// TIA Portal V18 export
FUNCTION "_motionLevel0_axis_main_in_cyclic_interrupt" : Void   // FC13, FBD
{ S7_Optimized_Access := 'TRUE' }
VERSION : 0.1
// stored: AutoNumber true, IsIECCheckEnabled false, SetENOAutomatically false, UDAEnableTagReadback false
   VAR_TEMP
      doors : Bool;
      "xray uses doors fwd closed mech" : Bool;
      "добавить блокировку вперед по световой завесе" : Bool;
      loc_dor_c_opn : Bool;
      loc_dor_c_cls : Bool;
      doorsWnOpnNAld : Bool;
      doorsWnClsNAld : Bool;
      ошибка_задания_искуственных_границ : Bool;
      динамическая_граница_y_rev : Real;
      динамическая_граница_y_fwd : Real;
      динамическая_граница_x_rev : Real;
      динамическая_граница_x_fwd : Real;
      манипулятор_не_мешает_дверям : Bool;
      doors_wnmanipulator : Bool;
   END_VAR
BEGIN

REGION Network 2
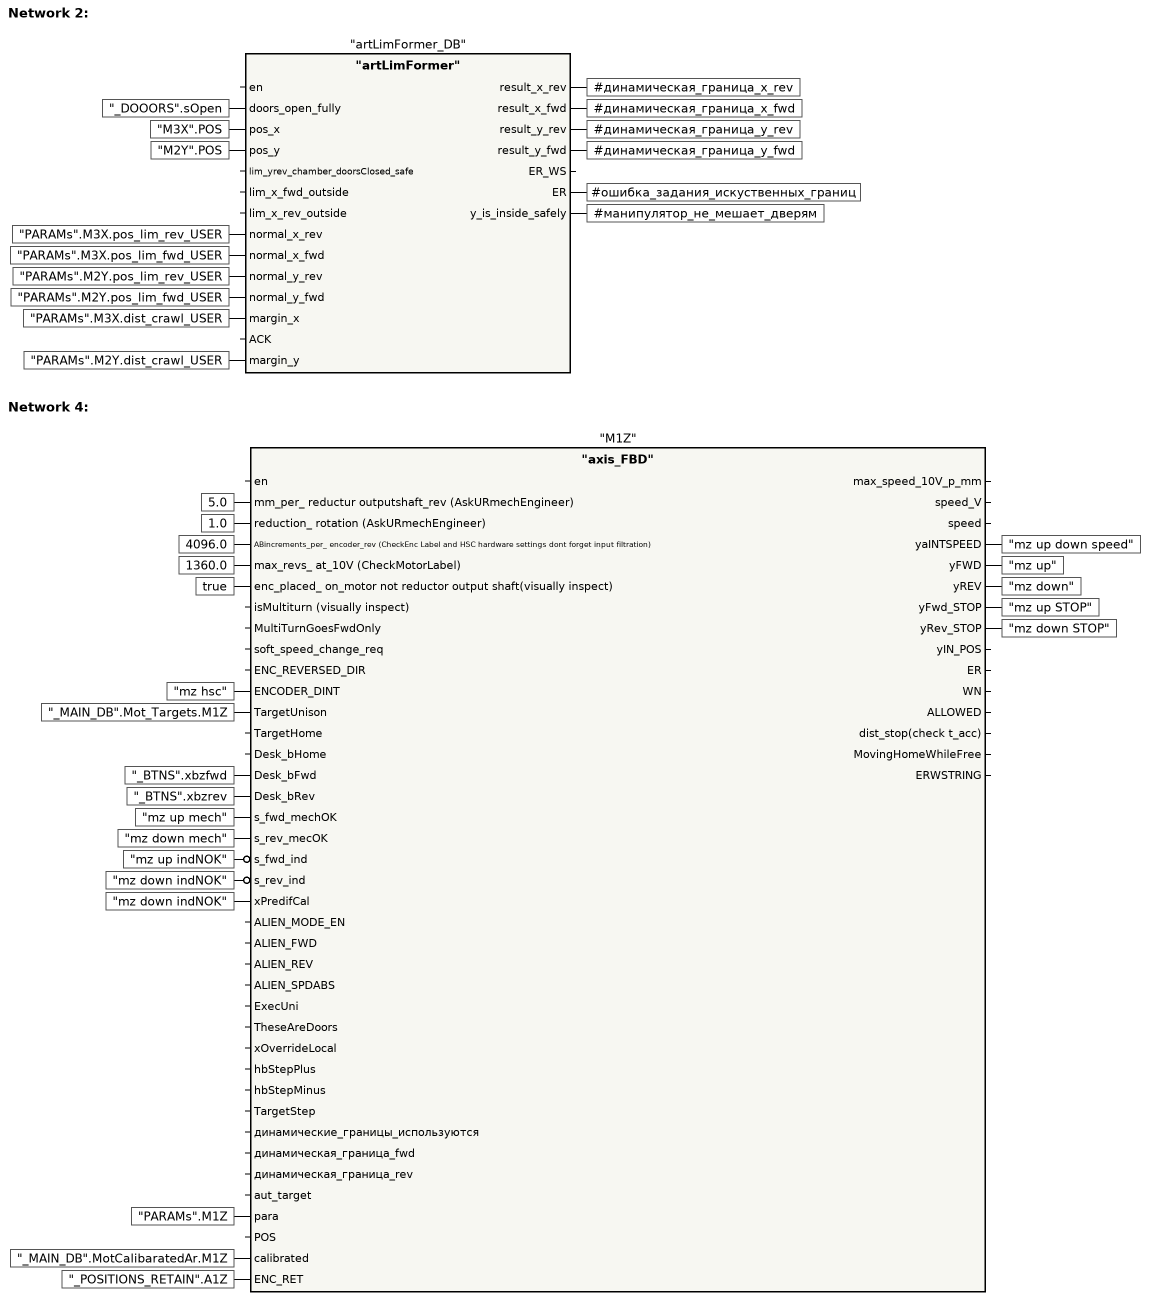
   "artLimFormer_DB"(doors_open_fully := "_DOOORS".sOpen,   // "artLimFormer"
                     pos_x := "M3X".POS,
                     pos_y := "M2Y".POS,
                     normal_x_rev := "PARAMs".M3X.pos_lim_rev_USER,
                     normal_x_fwd := "PARAMs".M3X.pos_lim_fwd_USER,
                     normal_y_rev := "PARAMs".M2Y.pos_lim_rev_USER,
                     normal_y_fwd := "PARAMs".M2Y.pos_lim_fwd_USER,
                     margin_x := "PARAMs".M3X.dist_crawl_USER,
                     margin_y := "PARAMs".M2Y.dist_crawl_USER,
                     result_x_rev => #динамическая_граница_x_rev,
                     result_x_fwd => #динамическая_граница_x_fwd,
                     result_y_rev => #динамическая_граница_y_rev,
                     result_y_fwd => #динамическая_граница_y_fwd,
                     ER => #ошибка_задания_искуственных_границ,
                     y_is_inside_safely => #манипулятор_не_мешает_дверям);
END_REGION

REGION Network 4
   "M1Z"("mm_per_ reductur outputshaft_rev (AskURmechEngineer)" := 5.0,   // "axis_FBD"
         "reduction_ rotation (AskURmechEngineer)" := 1.0,
         "ABincrements_per_ encoder_rev (CheckEnc Label and HSC hardware settings dont forget input filtration)" := 4096.0,
         "max_revs_ at_10V (CheckMotorLabel)" := 1360.0,
         "enc_placed_ on_motor not reductor output shaft(visually inspect)" := true,
         ENCODER_DINT := "mz hsc",
         TargetUnison := "_MAIN_DB".Mot_Targets.M1Z,
         Desk_bFwd := "_BTNS".xbzfwd,
         Desk_bRev := "_BTNS".xbzrev,
         s_fwd_mechOK := "mz up mech",
         s_rev_mecOK := "mz down mech",
         s_fwd_ind := NOT "mz up indNOK",
         s_rev_ind := NOT "mz down indNOK",
         xPredifCal := "mz down indNOK",
         para := "PARAMs".M1Z,
         calibrated := "_MAIN_DB".MotCalibaratedAr.M1Z,
         ENC_RET := "_POSITIONS_RETAIN".A1Z,
         yaINTSPEED => "mz up down speed",
         yFWD => "mz up",
         yREV => "mz down",
         yFwd_STOP => "mz up STOP",
         yRev_STOP => "mz down STOP");
END_REGION

REGION Network 5
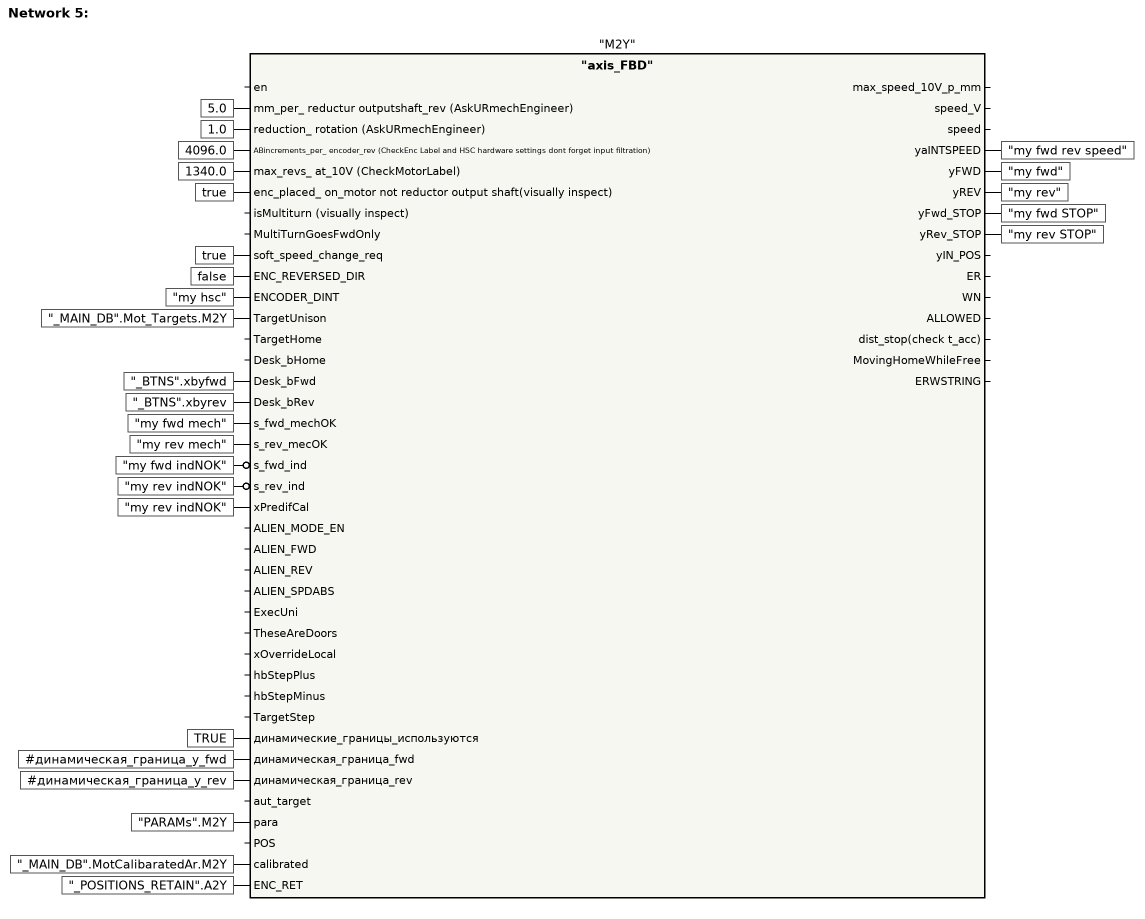
   "M2Y"("mm_per_ reductur outputshaft_rev (AskURmechEngineer)" := 5.0,   // "axis_FBD"
         "reduction_ rotation (AskURmechEngineer)" := 1.0,
         "ABincrements_per_ encoder_rev (CheckEnc Label and HSC hardware settings dont forget input filtration)" := 4096.0,
         "max_revs_ at_10V (CheckMotorLabel)" := 1340.0,
         "enc_placed_ on_motor not reductor output shaft(visually inspect)" := true,
         soft_speed_change_req := true,
         ENC_REVERSED_DIR := false,
         ENCODER_DINT := "my hsc",
         TargetUnison := "_MAIN_DB".Mot_Targets.M2Y,
         Desk_bFwd := "_BTNS".xbyfwd,
         Desk_bRev := "_BTNS".xbyrev,
         s_fwd_mechOK := "my fwd mech",
         s_rev_mecOK := "my rev mech",
         s_fwd_ind := NOT "my fwd indNOK",
         s_rev_ind := NOT "my rev indNOK",
         xPredifCal := "my rev indNOK",
         динамические_границы_используются := TRUE,
         динамическая_граница_fwd := #динамическая_граница_y_fwd,
         динамическая_граница_rev := #динамическая_граница_y_rev,
         para := "PARAMs".M2Y,
         calibrated := "_MAIN_DB".MotCalibaratedAr.M2Y,
         ENC_RET := "_POSITIONS_RETAIN".A2Y,
         yaINTSPEED => "my fwd rev speed",
         yFWD => "my fwd",
         yREV => "my rev",
         yFwd_STOP => "my fwd STOP",
         yRev_STOP => "my rev STOP");
END_REGION

REGION Network 6
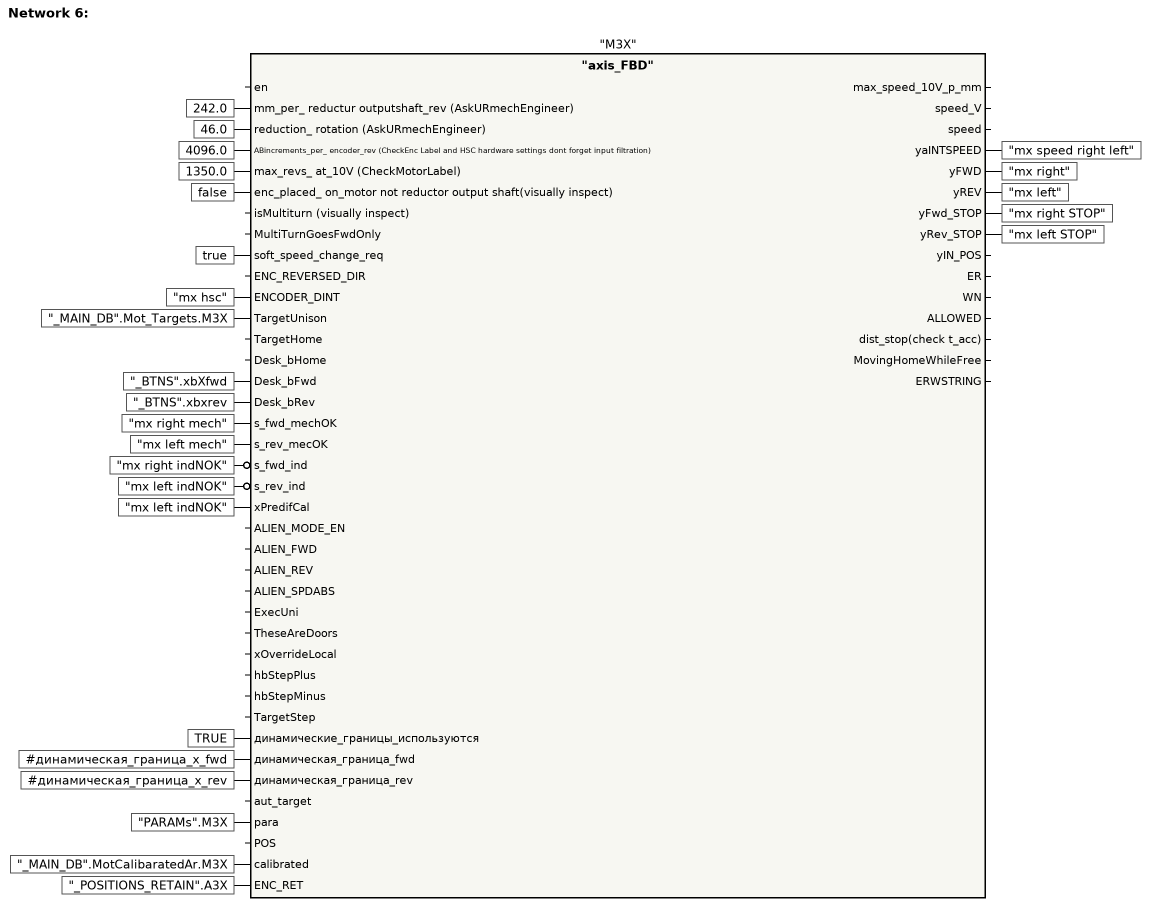
   "M3X"("mm_per_ reductur outputshaft_rev (AskURmechEngineer)" := 242.0,   // "axis_FBD"
         "reduction_ rotation (AskURmechEngineer)" := 46.0,
         "ABincrements_per_ encoder_rev (CheckEnc Label and HSC hardware settings dont forget input filtration)" := 4096.0,
         "max_revs_ at_10V (CheckMotorLabel)" := 1350.0,
         "enc_placed_ on_motor not reductor output shaft(visually inspect)" := false,
         soft_speed_change_req := true,
         ENCODER_DINT := "mx hsc",
         TargetUnison := "_MAIN_DB".Mot_Targets.M3X,
         Desk_bFwd := "_BTNS".xbXfwd,
         Desk_bRev := "_BTNS".xbxrev,
         s_fwd_mechOK := "mx right mech",
         s_rev_mecOK := "mx left mech",
         s_fwd_ind := NOT "mx right indNOK",
         s_rev_ind := NOT "mx left indNOK",
         xPredifCal := "mx left indNOK",
         динамические_границы_используются := TRUE,
         динамическая_граница_fwd := #динамическая_граница_x_fwd,
         динамическая_граница_rev := #динамическая_граница_x_rev,
         para := "PARAMs".M3X,
         calibrated := "_MAIN_DB".MotCalibaratedAr.M3X,
         ENC_RET := "_POSITIONS_RETAIN".A3X,
         yaINTSPEED => "mx speed right left",
         yFWD => "mx right",
         yREV => "mx left",
         yFwd_STOP => "mx right STOP",
         yRev_STOP => "mx left STOP");
END_REGION

REGION Network 7
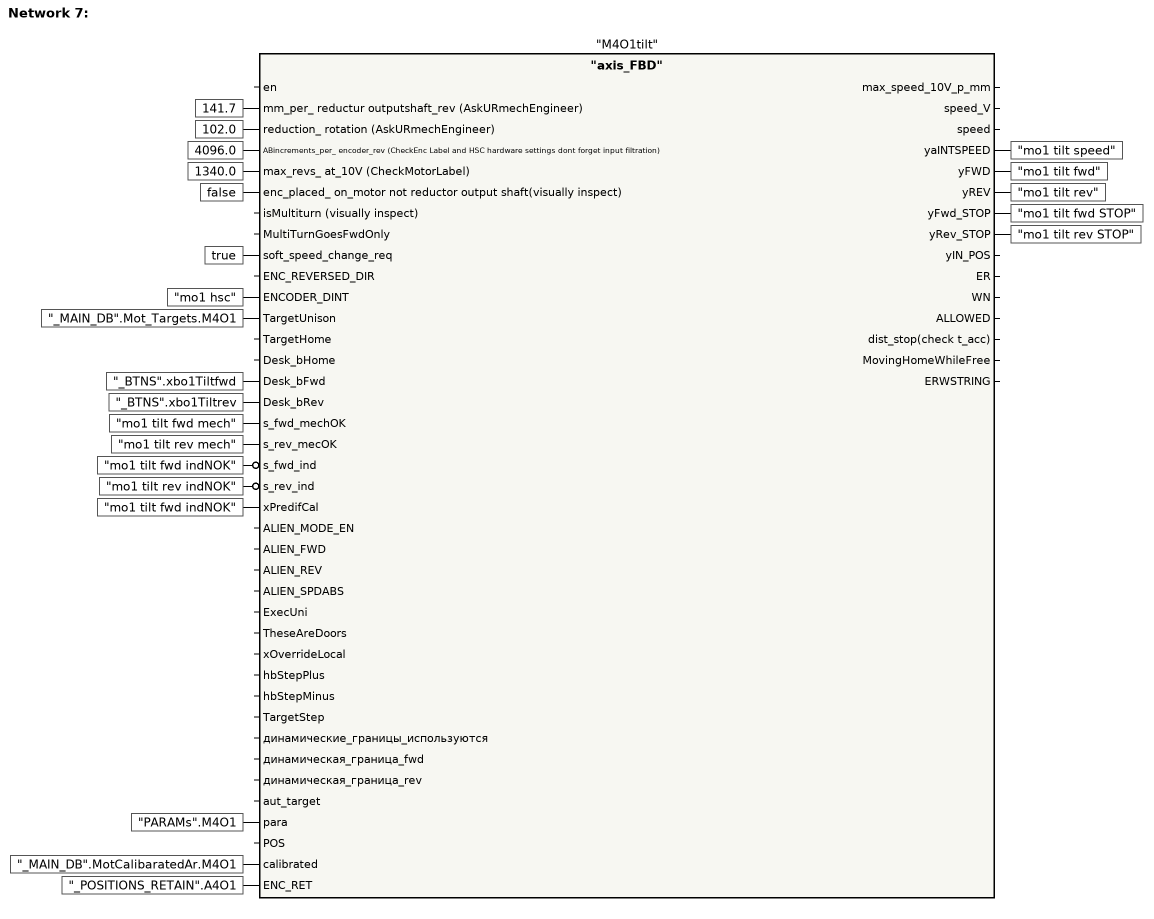
   "M4O1tilt"("mm_per_ reductur outputshaft_rev (AskURmechEngineer)" := 141.7,   // "axis_FBD"
              "reduction_ rotation (AskURmechEngineer)" := 102.0,
              "ABincrements_per_ encoder_rev (CheckEnc Label and HSC hardware settings dont forget input filtration)" := 4096.0,
              "max_revs_ at_10V (CheckMotorLabel)" := 1340.0,
              "enc_placed_ on_motor not reductor output shaft(visually inspect)" := false,
              soft_speed_change_req := true,
              ENCODER_DINT := "mo1 hsc",
              TargetUnison := "_MAIN_DB".Mot_Targets.M4O1,
              Desk_bFwd := "_BTNS".xbo1Tiltfwd,
              Desk_bRev := "_BTNS".xbo1Tiltrev,
              s_fwd_mechOK := "mo1 tilt fwd mech",
              s_rev_mecOK := "mo1 tilt rev mech",
              s_fwd_ind := NOT "mo1 tilt fwd indNOK",
              s_rev_ind := NOT "mo1 tilt rev indNOK",
              xPredifCal := "mo1 tilt fwd indNOK",
              para := "PARAMs".M4O1,
              calibrated := "_MAIN_DB".MotCalibaratedAr.M4O1,
              ENC_RET := "_POSITIONS_RETAIN".A4O1,
              yaINTSPEED => "mo1 tilt speed",
              yFWD => "mo1 tilt fwd",
              yREV => "mo1 tilt rev",
              yFwd_STOP => "mo1 tilt fwd STOP",
              yRev_STOP => "mo1 tilt rev STOP");
END_REGION

REGION Network 8
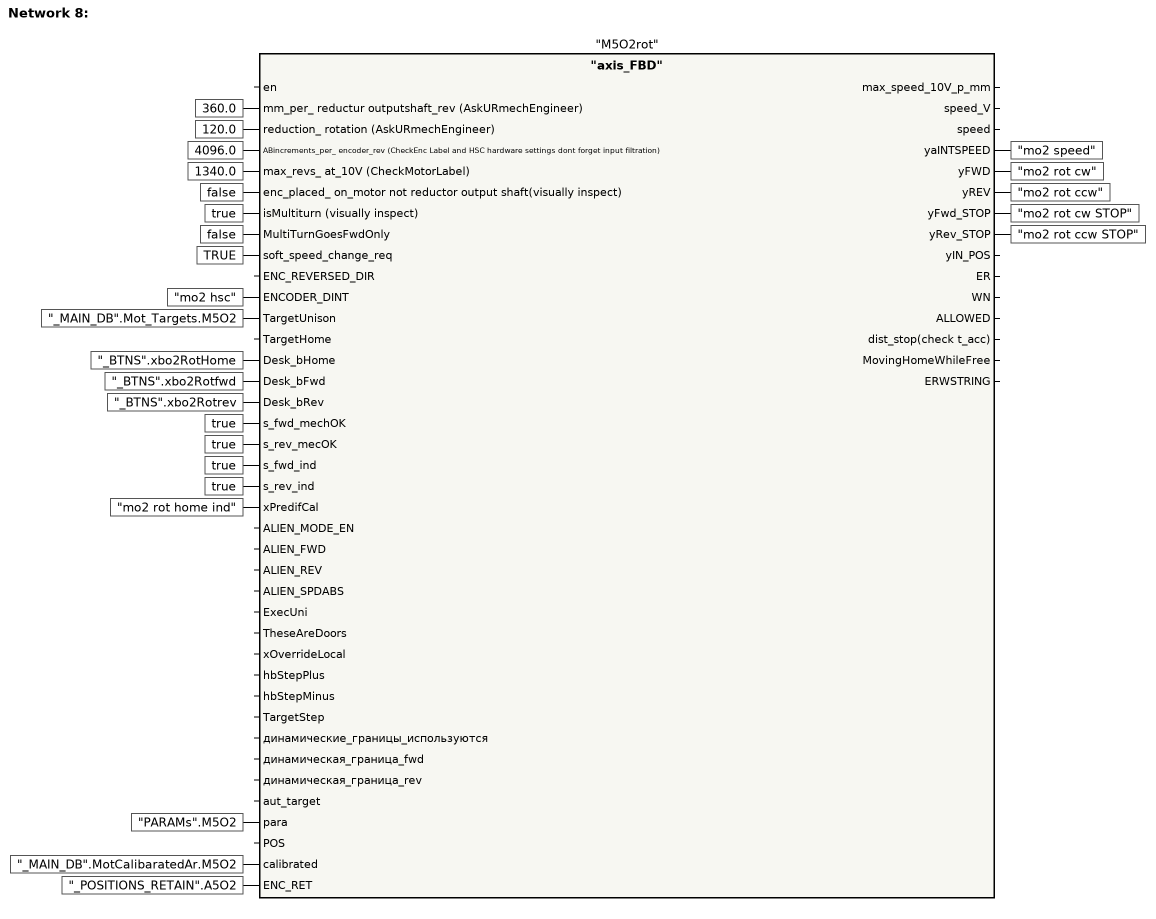
   "M5O2rot"("mm_per_ reductur outputshaft_rev (AskURmechEngineer)" := 360.0,   // "axis_FBD"
             "reduction_ rotation (AskURmechEngineer)" := 120.0,
             "ABincrements_per_ encoder_rev (CheckEnc Label and HSC hardware settings dont forget input filtration)" := 4096.0,
             "max_revs_ at_10V (CheckMotorLabel)" := 1340.0,
             "enc_placed_ on_motor not reductor output shaft(visually inspect)" := false,
             "isMultiturn (visually inspect)" := true,
             MultiTurnGoesFwdOnly := false,
             soft_speed_change_req := TRUE,
             ENCODER_DINT := "mo2 hsc",
             TargetUnison := "_MAIN_DB".Mot_Targets.M5O2,
             Desk_bHome := "_BTNS".xbo2RotHome,
             Desk_bFwd := "_BTNS".xbo2Rotfwd,
             Desk_bRev := "_BTNS".xbo2Rotrev,
             s_fwd_mechOK := true,
             s_rev_mecOK := true,
             s_fwd_ind := true,
             s_rev_ind := true,
             xPredifCal := "mo2 rot home ind",
             para := "PARAMs".M5O2,
             calibrated := "_MAIN_DB".MotCalibaratedAr.M5O2,
             ENC_RET := "_POSITIONS_RETAIN".A5O2,
             yaINTSPEED => "mo2 speed",
             yFWD => "mo2 rot cw",
             yREV => "mo2 rot ccw",
             yFwd_STOP => "mo2 rot cw STOP",
             yRev_STOP => "mo2 rot ccw STOP");
END_REGION

REGION Network 9
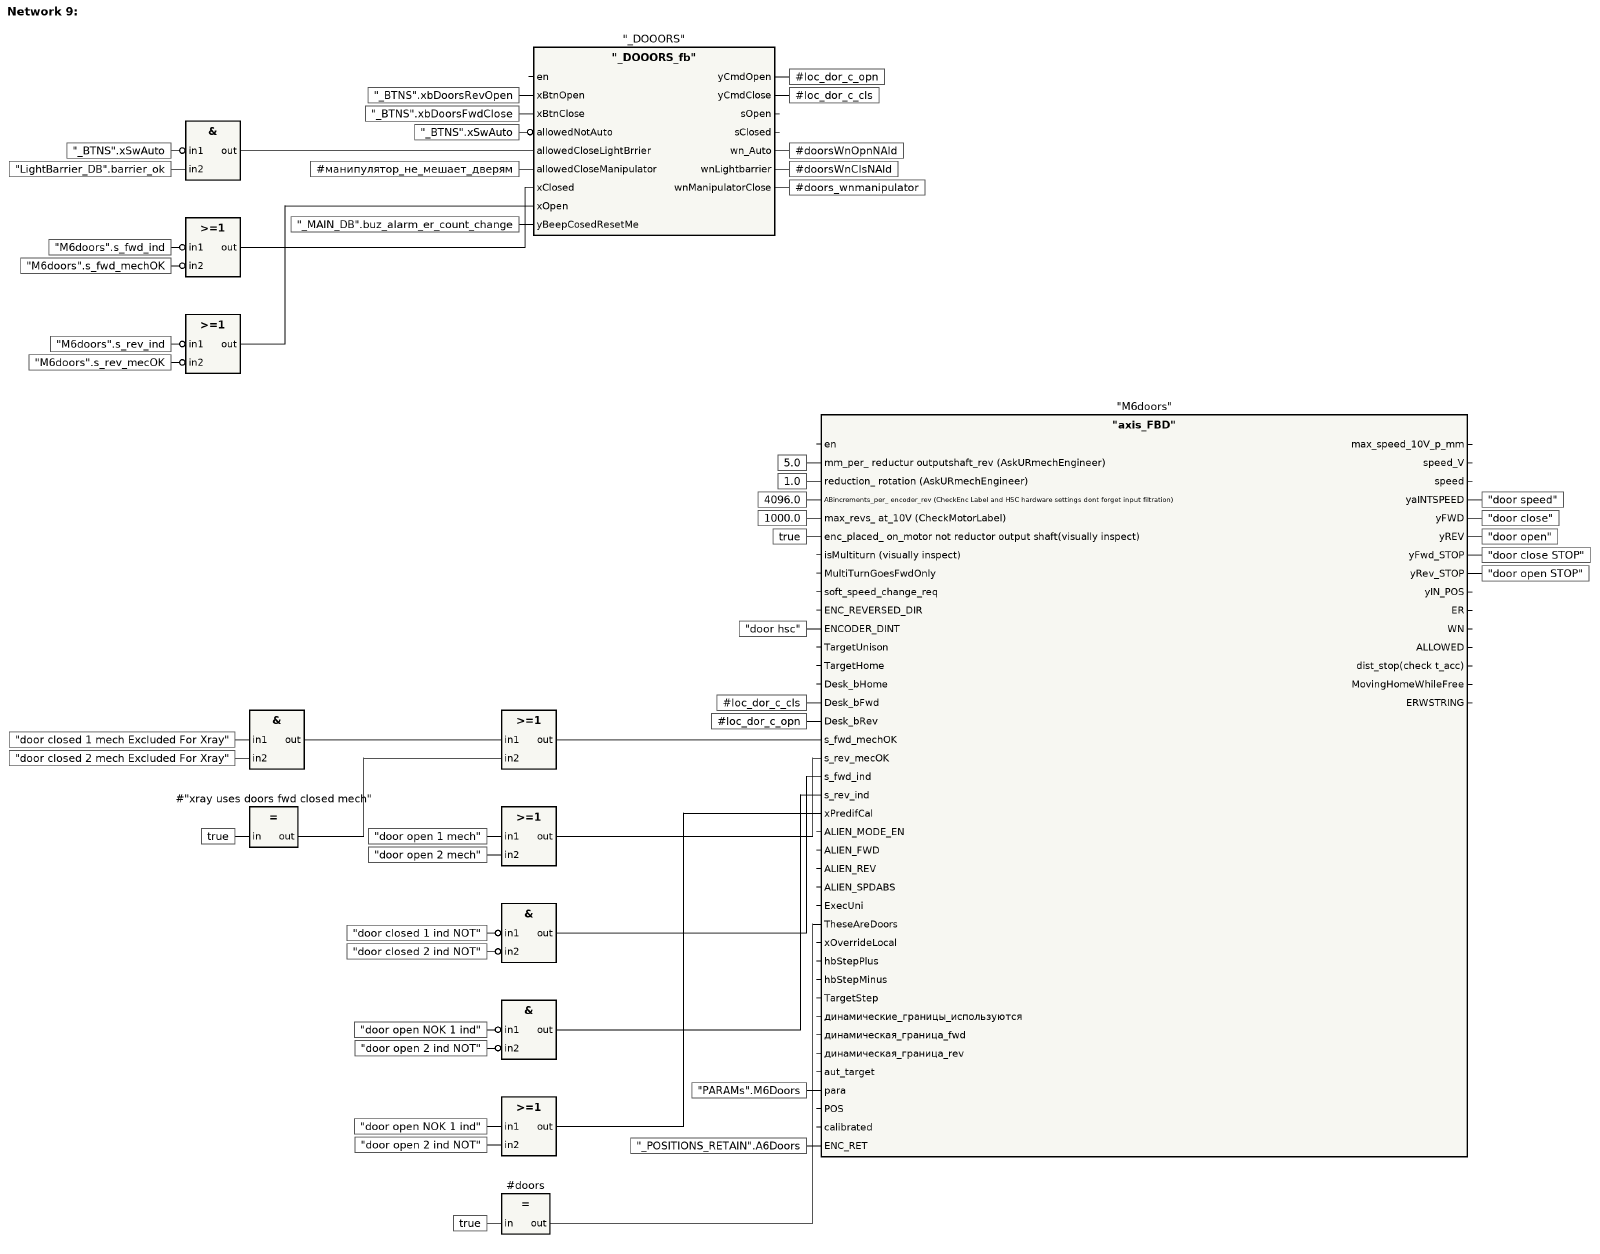
   "_DOOORS"(xBtnOpen := "_BTNS".xbDoorsRevOpen,   // "_DOOORS_fb"
             xBtnClose := "_BTNS".xbDoorsFwdClose,
             allowedNotAuto := NOT "_BTNS".xSwAuto,
             allowedCloseLightBrrier := NOT "_BTNS".xSwAuto AND "LightBarrier_DB".barrier_ok,
             allowedCloseManipulator := #манипулятор_не_мешает_дверям,
             xClosed := NOT "M6doors".s_fwd_ind OR NOT "M6doors".s_fwd_mechOK,
             xOpen := NOT "M6doors".s_rev_ind OR NOT "M6doors".s_rev_mecOK,
             yBeepCosedResetMe := "_MAIN_DB".buz_alarm_er_count_change,
             yCmdOpen => #loc_dor_c_opn,
             yCmdClose => #loc_dor_c_cls,
             wn_Auto => #doorsWnOpnNAld,
             wnLightbarrier => #doorsWnClsNAld,
             wnManipulatorClose => #doors_wnmanipulator);
   #"xray uses doors fwd closed mech" := true;
   #doors := true;
   "M6doors"("mm_per_ reductur outputshaft_rev (AskURmechEngineer)" := 5.0,   // "axis_FBD"
             "reduction_ rotation (AskURmechEngineer)" := 1.0,
             "ABincrements_per_ encoder_rev (CheckEnc Label and HSC hardware settings dont forget input filtration)" := 4096.0,
             "max_revs_ at_10V (CheckMotorLabel)" := 1000.0,
             "enc_placed_ on_motor not reductor output shaft(visually inspect)" := true,
             ENCODER_DINT := "door hsc",
             Desk_bFwd := #loc_dor_c_cls,
             Desk_bRev := #loc_dor_c_opn,
             s_fwd_mechOK := ("door closed 1 mech Excluded For Xray" AND "door closed 2 mech Excluded For Xray") OR true,
             s_rev_mecOK := "door open 1 mech" OR "door open 2 mech",
             s_fwd_ind := NOT "door closed 1 ind NOT" AND NOT "door closed 2 ind NOT",
             s_rev_ind := NOT "door open NOK 1 ind" AND NOT "door open 2 ind NOT",
             xPredifCal := "door open NOK 1 ind" OR "door open 2 ind NOT",
             TheseAreDoors := true,
             para := "PARAMs".M6Doors,
             ENC_RET := "_POSITIONS_RETAIN".A6Doors,
             yaINTSPEED => "door speed",
             yFWD => "door close",
             yREV => "door open",
             yFwd_STOP => "door close STOP",
             yRev_STOP => "door open STOP");
END_REGION

REGION Network 10
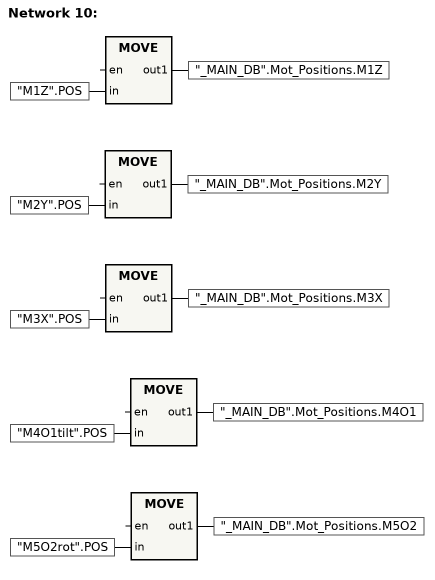
   "_MAIN_DB".Mot_Positions.M1Z := "M1Z".POS;
   "_MAIN_DB".Mot_Positions.M2Y := "M2Y".POS;
   "_MAIN_DB".Mot_Positions.M3X := "M3X".POS;
   "_MAIN_DB".Mot_Positions.M4O1 := "M4O1tilt".POS;
   "_MAIN_DB".Mot_Positions.M5O2 := "M5O2rot".POS;
END_REGION

REGION Network 11
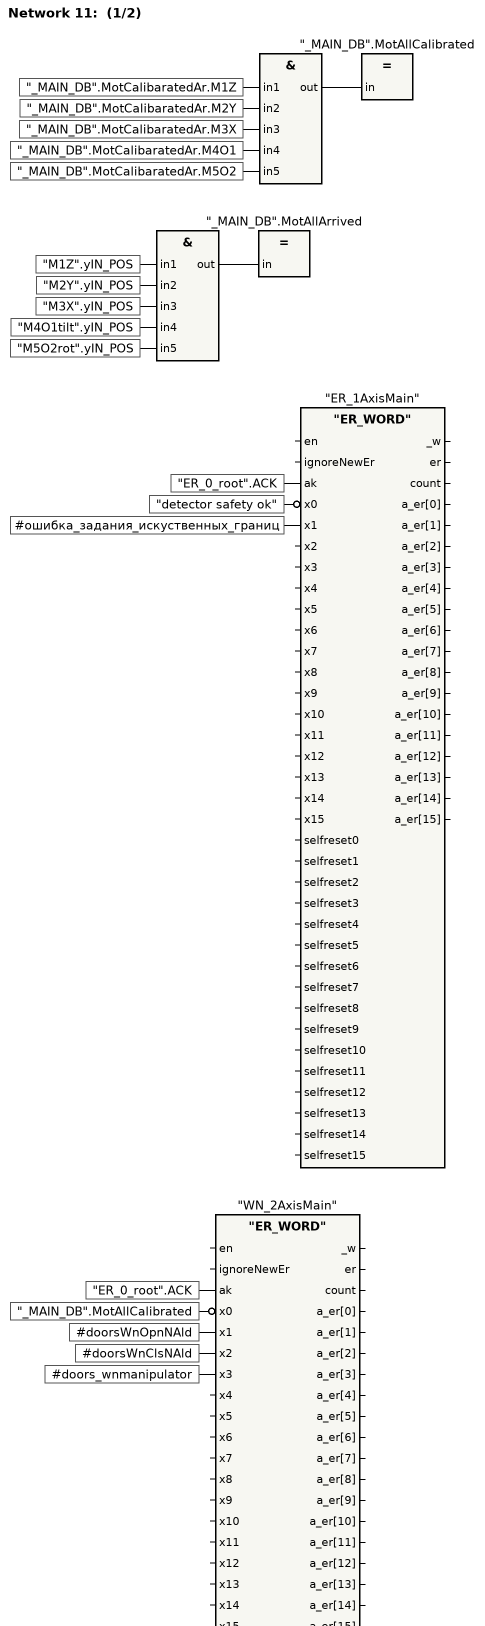
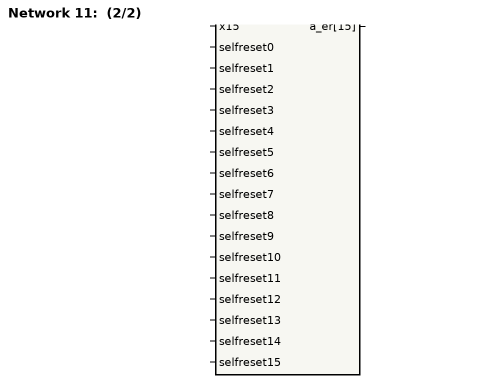
   "_MAIN_DB".MotAllCalibrated := "_MAIN_DB".MotCalibaratedAr.M1Z AND "_MAIN_DB".MotCalibaratedAr.M2Y AND "_MAIN_DB".MotCalibaratedAr.M3X AND "_MAIN_DB".MotCalibaratedAr.M4O1 AND "_MAIN_DB".MotCalibaratedAr.M5O2;
   "_MAIN_DB".MotAllArrived := "M1Z".yIN_POS AND "M2Y".yIN_POS AND "M3X".yIN_POS AND "M4O1tilt".yIN_POS AND "M5O2rot".yIN_POS;
   "ER_1AxisMain"(ak := "ER_0_root".ACK,   // "ER_WORD"
                  x0 := NOT "detector safety ok",
                  x1 := #ошибка_задания_искуственных_границ);
   "WN_2AxisMain"(ak := "ER_0_root".ACK,   // "ER_WORD"
                  x0 := NOT "_MAIN_DB".MotAllCalibrated,
                  x1 := #doorsWnOpnNAld,
                  x2 := #doorsWnClsNAld,
                  x3 := #doors_wnmanipulator);
END_REGION
END_FUNCTION
